PROGRAM MAIN
VAR
END_VAR

P_COMMIT1();

END_PROGRAM

(* stored: Version 1.1.0.1, ProductVersion 3.1.4024.12
   POU MAIN: Id {bb454c8f-4521-4fb5-a70c-622ab5d5fe57}, SpecialFunc None *)
